FUNCTION_BLOCK FB_EventLogger
VAR
	bBoolean : BOOL := FALSE;
	
	// Event example
	eEventType1 : E_EventType := E_EventType.Alarm;
	eEventSeverity1 : TcEventSeverity.Error;
	nEventIdentity1 : UDINT := 1;
	sEventText1 : STRING(255) := "This is an example";
	
	fbCsvPersistantEventStorage : FB_CsvPersistantEventStorage;
	fbEventLogger : FB_EventLogger(fbCsvPersistantEventStorage);
END_VAR

//Example of event
IF bBoolean THEN
	EventLogger.AddEvent(eEventType1, eEventSeverity1, nEventIdentity1, sEventText1);
END_IF

fbCsvPersistantEventStorage();

END_FUNCTION_BLOCK

(* stored: Version 1.1.0.1
   POU FB_EventLogger: Id {c3e5ec1d-5cfb-4980-a176-b11a253ef344}, SpecialFunc None *)
